(* CoDeSys 2.3 export: ACTUATOR_3P.EXP *)

(* POU actuators/ACTUATOR_3P, ST *)
FUNCTION_BLOCK ACTUATOR_3P
VAR_INPUT
	IN : BYTE;
	TEST : BOOL;
	ARE : BOOL := TRUE;
	END_POS : BOOL;
END_VAR
VAR_INPUT CONSTANT
	T_RUN : TIME := t#10s; (*Время открытия клапана*)
	T_EXT : TIME := T#1s;
	T_CAL : TIME := t#1s;
	T_DIAG : TIME := T#30d;
	SWITCH_AVAIL : BOOL := TRUE; (*False включить диагностику*)

END_VAR
VAR_IN_OUT

END_VAR
VAR_OUTPUT
	OUT1 : BOOL;
	OUT2 : BOOL;
	POS : BYTE;
	ERROR : BOOL;
	STATUS : BYTE;
END_VAR
VAR
	ramp : _RMP_NEXT;
	tx : TIME ;
	next_cal : TIME;
	next_diag : TIME;
	last: TIME;
	start: TIME;
	ARX : BOOL:=FALSE;
END_VAR


(*
version 2.0	28. jan 2010
programmer 	hugo
tested by		oscat

actuator_3P is an interface for a 3 point actuator.
a 3P actuator is a motor with 2 directions that drives a valve or flap. the position of the valve or flap is controlled by runtime of the motor foreward or backward.
the available inputs are:
IN specifies the position of the actuator, 0 = 0% and 255 = 100%.
an END_POS input is available for an end_pos switch, this switch indicates the valve or flap to be at either 0% or 100%
a TEST input can at any time start a diag cycle which turns the motor towards the 0% position, then measures the runtime to 100% and then the runtime to 0%
these runtimes are stored and used for absolute positioning of the motor during normal operation. this feature is only avaliable with an END_POS switch connected to the input.
a setup variable T_DIAG can be used to specify how often the actuator repeates this auto_diag cycle automatically.
at power on a diag cycle is perfomed automatically.
a time of 0 for T_DIAG means auto diag is never performed.

the outputs out1 and out2 are for the two directions of the motor.
a pos output indicates the simulated position of the actuator during operation.
a error output is activated when the specified max_runtime is reached by any direction during debug without an end_switch to become active.
also when the up and down direction differs by more then 10% the error output is set.

for absolute positioning accuracy the actuator has a setup variable "cal_runtime" if this is set the actuator measures the total runtime of the motors and when this 
cal_runtime is exceeded it resets the actuator to 0% position and sets the output again to assure absolute accuracy.

test and calibration can be shut off by setting the appropriate values to 0.
a switch_available setup variable specifies if end_pos switches are available.

*)
(* read system timer *)
tx := DWORD_TO_TIME(T_PLC_MS());

(* check test input *)
IF TEST THEN
	status := 103;
	start := tx;
	(*ARX := TRUE; *)
END_IF;

CASE status OF
	0:	(* power on setup *)
		IF ARE AND NOT ARX THEN
			status := 103;
			start := tx;
			(*ARX := TRUE; *)
		END_IF;

	100:	(* normal operation *)
		(* check for auto diagnostics *)
		IF T_DIAG > T#0s AND tx > next_diag AND ARE AND NOT ARX THEN
				status := 103;
				start := tx;
				(*ARX := TRUE; *)

		(* check for auto calibration *)
		ELSIF T_CAL > T#0s AND tx > next_cal AND ARE AND NOT ARX THEN
			IF pos > BYTE#127THEN
				OUT1 := TRUE;
				OUT2 := FALSE;
				ramp.IN := 255;
				(*ARX := TRUE; *)
			ELSE
				OUT1 := FALSE;
				OUT2 := TRUE;
				ramp.IN := 0;
				(*ARX := TRUE; *)
			END_IF;
			status := 101;
			start := tx;
		ELSE
			(* increment next_cal if not active *)
			IF NOT(OUT1 OR OUT2) THEN next_cal := next_cal + (tx-last); END_IF;
			(* set ramp generator to IN *)
			ramp.IN := IN;
		END_IF;

	101:	(* calibrate *)
		IF tx - start < T_EXT THEN
			next_cal := tx + T_CAL;
		ELSIF SWITCH_AVAIL AND END_POS THEN
			STATUS := 100;
			(*ARX := FALSE; *)
		ELSIF tx - start > T_EXT + T_RUN THEN
			ERROR := SWITCH_AVAIL;
			(*ARX := FALSE; *)
		END_IF;

	103:	(* diagnostics up*)
		(* run up for T_ext *)
		IF tx - start < T_EXT THEN
			ERROR := FALSE;
			ramp.TR := T_RUN;
			ramp.TF := T_RUN;
			OUT1 := TRUE;
			OUT2 := FALSE;
			ramp.IN := 255;
		ELSIF SWITCH_AVAIL AND END_POS THEN
			ramp.TR := tx - start;
			STATUS := 104;
		ELSIF tx - start > T_EXT + T_RUN THEN
			ERROR := SWITCH_AVAIL;
			STATUS := 104;
			start := tx;
		END_IF;

	104:	(* diagnostics dn*)
		IF tx - start < T_ext THEN
			OUT1 := FALSE;
			OUT2 := TRUE;
			ramp.IN := 0;
			next_diag := tx + T_DIAG;
		ELSIF SWITCH_AVAIL AND END_POS THEN
			ramp.TR := tx - start;
			(* check if runtimes differ by more than 10% *)
			IF DINT_TO_TIME(ABS(TIME_TO_DINT(ramp.TR) - TIME_TO_DINT(ramp.TF))*10) > T_RUN THEN error := TRUE; END_IF;
			STATUS := 100;
			(*ARX := FALSE; *)
			next_cal := tx + T_CAL;
		ELSIF tx - start > T_EXT + T_RUN THEN
			IF SWITCH_AVAIL THEN ERROR := TRUE; END_IF;
			STATUS := 100;
			(*ARX := FALSE; *)
			next_CAL := tx + T_CAL;
		END_IF;
END_CASE;

(* internal flap simulation and output activation *)
ramp(OUT := POS);
IF STATUS = 100 THEN
	OUT1 := ramp.UP;
	OUT2 := ramp.DN;
END_IF;

(* adjust position if end switch is active *)
IF SWITCH_AVAIL AND END_POS THEN
	POS := SEL(POS > 127, 0, 255);
	next_cal := tx + T_CAL;
END_IF;

(* set last to tx for next cycle *)
last := tx;



(* revision history

hm	19. oct 2006	rev 1.1
	added security checks for end_switch to avoid overrun of the end_switch, hans

hm	23. jan 2007	rev 1.2
	deleted unused variables force_on and force_off

hm	15. sep 2007	 rev 1.3
	replaced Time() with T_PLC_MS for compatibility and performance reasons

hm	28. jan 2010	rev 2.0
	new code and new features

*)
END_FUNCTION_BLOCK
